// TIA Portal V20 export
TYPE "typeEm5MonitoringSoftCam"
// stored: Access Published, Namespace Unit1
   STRUCT
      manualInputPp { ExternalWritable := 'False'} : "LER_typeSoftCamRelation";
      magazineLift { ExternalWritable := 'False'} : "LER_typeSoftCamRelation";
   END_STRUCT;
   // // manualInputPp.posistion0 : LoadingPos
   // // manualInputPp.posistion1 : UnLoadingPos
   // // magazineLift.posistion0 : HomePos
   // // magazineLift.posistion1 : WorkPos
END_TYPE
